// User intent pass-through into the shadow operational layer
GVL_COMMAND_SHADOW.G_Gate_Open := GVL_INTENT_USER.I_Gate_Open_Request;
GVL_COMMAND_SHADOW.G_Wicket_Open := GVL_INTENT_USER.I_Wicket_Open_Request;
GVL_COMMAND_SHADOW.G_Lock_1_Open := GVL_INTENT_USER.I_Lock_1_Open_Request;
GVL_COMMAND_SHADOW.G_Lock_1_Close := GVL_INTENT_USER.I_Lock_1_Close_Request;
GVL_COMMAND_SHADOW.G_Lock_2_Open := GVL_INTENT_USER.I_Lock_2_Open_Request;
GVL_COMMAND_SHADOW.G_Lock_2_Close := GVL_INTENT_USER.I_Lock_2_Close_Request;

// Safety and system arbitration into the shadow operational layer
IF GVL_INTENT_SAFETY.I_Fire_Alarm_Active THEN
    GVL_COMMAND_SHADOW.G_Boiler_Stop := TRUE;
    GVL_COMMAND_SHADOW.G_Vent_Stop := TRUE;
    GVL_COMMAND_SHADOW.G_Lock_1_Open := TRUE;
    GVL_COMMAND_SHADOW.G_Lock_2_Open := TRUE;
END_IF;

IF GVL_INTENT_SAFETY.I_Gas_Close_Required THEN
    GVL_COMMAND_SHADOW.G_Gas_Valve_Close := TRUE;
    GVL_COMMAND_SHADOW.G_Boiler_Stop := TRUE;
END_IF;

IF GVL_INTENT_SAFETY.I_Vent_Force_PV3_Boost THEN
    GVL_COMMAND_SHADOW.G_Vent_PV3_Boost := TRUE;
END_IF;

IF GVL_INTENT_SAFETY.I_Vent_Force_Supply_100 THEN
    GVL_COMMAND_SHADOW.G_Supply_100_Req := TRUE;
END_IF;

IF GVL_INTENT_SAFETY.I_Vent_Force_Supply_80 THEN
    GVL_COMMAND_SHADOW.G_Supply_80_Req := TRUE;
END_IF;

IF GVL_INTENT_SAFETY.I_Vent_Stop_Required THEN
    GVL_COMMAND_SHADOW.G_Vent_Stop := TRUE;
END_IF;

IF GVL_INTENT_SYSTEM.I_Mode_Degraded_Active THEN
    GVL_COMMAND_SHADOW.G_Supply_80_Req := TRUE;
END_IF;

IF GVL_INTENT_SAFETY.I_Water_Main_Close_Required THEN
    GVL_COMMAND_SHADOW.G_Close_Valve_35 := TRUE;
    GVL_COMMAND_SHADOW.G_Close_Valve_36 := TRUE;
END_IF;

FOR L_i := 1 TO 32 DO
    IF GVL_INTENT_SAFETY.I_Water_Zone_Close_Required[L_i] THEN
        ;
    END_IF;
END_FOR;
          
END_PROGRAM

PROGRAM PRG_System_Test_Harness
  VAR
    L_i : INT;
    L_j : INT;
    L_Used : REAL;
    L_HP_Used : REAL;
    L_HP_Manifold_Adjusted : ARRAY[1..GVL_CONSTANTS.C_MAX_MANIFOLDS] OF INT;
    fbDecisionTest : FB_Heating_Decision_Context;
    fbDecisionHP : FB_Heating_Decision_Context;
    fbTestResult : FB_Test_Result_Handler;
    fbTrace : FB_Trace_Logger;
  END_VAR

            IF NOT GVL_TEST.G_Test_Enable THEN
    RETURN;
END_IF;

GVL_TEST.G_Test_Total_Checks := 0;
GVL_TEST.G_Test_Failed_Checks := 0;
GVL_TEST.G_Test_Passed := TRUE;
GVL_TEST.G_Test_Last_Failure_Index := 0;
GVL_TEST.G_Test_Last_Failure_Code := 0;

// Reset transient failure flags for this scan
GVL_TEST.G_Diagnostics_Duplicate_Event_Found := FALSE;
GVL_TEST.G_Diagnostics_Count_Out_Of_Range := FALSE;
GVL_TEST.G_Heating_Allocation_Budget_Exceeded := FALSE;
GVL_TEST.G_Heating_Allocation_Enabled_Not_Allowed := FALSE;
GVL_TEST.G_Safety_Latched_Without_Intent := FALSE;
GVL_TEST.G_HP_Adjusted_Priority_Lower_Bound_Violation := FALSE;
GVL_TEST.G_HP_Adjusted_Allocation_Budget_Exceeded := FALSE;
GVL_TEST.G_HP_Adjusted_Allocation_Enabled_Not_Allowed := FALSE;
GVL_TEST.G_HP_Guest_Preheat_Config_Out_Of_Range := FALSE;

// =========================
// TEST 1: Diagnostics count bounds
// =========================
GVL_TEST.G_Test_Total_Checks := GVL_TEST.G_Test_Total_Checks + 1;
IF (GVL_STATUS.G_Diagnostics_Count < 0) OR (GVL_STATUS.G_Diagnostics_Count > 50) THEN
    GVL_TEST.G_Diagnostics_Count_Out_Of_Range := TRUE;
    GVL_TEST.G_Test_Failed_Checks := GVL_TEST.G_Test_Failed_Checks + 1;
    GVL_TEST.G_Test_Passed := FALSE;
    GVL_TEST.G_Test_Last_Failure_Index := 1;
    GVL_TEST.G_Test_Last_Failure_Code := 1001;
END_IF;

// =========================
// TEST 2: Diagnostics duplicates
// =========================
GVL_TEST.G_Test_Total_Checks := GVL_TEST.G_Test_Total_Checks + 1;
FOR L_i := 1 TO GVL_STATUS.G_Diagnostics_Count DO
    FOR L_j := L_i + 1 TO GVL_STATUS.G_Diagnostics_Count DO
        IF (GVL_STATUS.G_Diagnostics_Events[L_i].Code = GVL_STATUS.G_Diagnostics_Events[L_j].Code) AND
           (GVL_STATUS.G_Diagnostics_Events[L_i].Source = GVL_STATUS.G_Diagnostics_Events[L_j].Source) THEN
            GVL_TEST.G_Diagnostics_Duplicate_Event_Found := TRUE;
            GVL_TEST.G_Test_Failed_Checks := GVL_TEST.G_Test_Failed_Checks + 1;
            GVL_TEST.G_Test_Passed := FALSE;
            GVL_TEST.G_Test_Last_Failure_Index := 2;
            GVL_TEST.G_Test_Last_Failure_Code := 1002;
        END_IF;
    END_FOR;
END_FOR;

// =========================
// TEST 3: Base heating decision consistency
// =========================
GVL_TEST.G_Test_Total_Checks := GVL_TEST.G_Test_Total_Checks + 1;
fbDecisionTest(
    VI_Manifold_Pump_In_Service := GVL_CONFIG.G_Manifold_Pump_In_Service,
    VI_Manifold_Pressure_Fault := GVL_STATUS.G_Diagnostics.Manifold_Pressure_Fault,
    VI_Manifold_Current_Fault := GVL_STATUS.G_Diagnostics.Manifold_Current_Fault,
    VI_Manifold_Thermal_Weight := GVL_CONFIG.G_Manifold_Thermal_Weight,
    VI_Manifold_Priority := GVL_CONFIG.G_Manifold_Priority,
    VI_Max_Thermal_Budget := GVL_CONFIG.G_Max_Thermal_Budget
);

L_Used := 0.0;
FOR L_i := 1 TO GVL_CONSTANTS.C_MAX_MANIFOLDS DO
    IF fbDecisionTest.VO_Manifold_Enabled[L_i] AND (NOT fbDecisionTest.VO_Manifold_Allowed[L_i]) THEN
        GVL_TEST.G_Heating_Allocation_Enabled_Not_Allowed := TRUE;
        GVL_TEST.G_Test_Failed_Checks := GVL_TEST.G_Test_Failed_Checks + 1;
        GVL_TEST.G_Test_Passed := FALSE;
        GVL_TEST.G_Test_Last_Failure_Index := 3;
        GVL_TEST.G_Test_Last_Failure_Code := 1003;
    END_IF;

    IF fbDecisionTest.VO_Manifold_Enabled[L_i] THEN
        L_Used := L_Used + GVL_CONFIG.G_Manifold_Thermal_Weight[L_i];
    END_IF;
END_FOR;

IF L_Used > (GVL_CONFIG.G_Max_Thermal_Budget + 0.001) THEN
    GVL_TEST.G_Heating_Allocation_Budget_Exceeded := TRUE;
    GVL_TEST.G_Test_Failed_Checks := GVL_TEST.G_Test_Failed_Checks + 1;
    GVL_TEST.G_Test_Passed := FALSE;
    GVL_TEST.G_Test_Last_Failure_Index := 3;
    GVL_TEST.G_Test_Last_Failure_Code := 1004;
END_IF;

// =========================
// TEST 4: Safety latch consistency
// =========================
GVL_TEST.G_Test_Total_Checks := GVL_TEST.G_Test_Total_Checks + 1;
IF GVL_STATE.G_Safety_Gas_Latched AND (NOT GVL_INTENT_SAFETY.I_Gas_Alarm_Active) THEN
    GVL_TEST.G_Safety_Latched_Without_Intent := TRUE;
    GVL_TEST.G_Test_Failed_Checks := GVL_TEST.G_Test_Failed_Checks + 1;
    GVL_TEST.G_Test_Passed := FALSE;
    GVL_TEST.G_Test_Last_Failure_Index := 4;
    GVL_TEST.G_Test_Last_Failure_Code := 1005;
END_IF;

// =========================
// TEST 5: HP policy adjusted priority
// =========================
GVL_TEST.G_Test_Total_Checks := GVL_TEST.G_Test_Total_Checks + 1;

IF (GVL_HEATING_POLICY_CONFIG.G_Guest_Preheat_Priority_Boost < 0) OR (GVL_HEATING_POLICY_CONFIG.G_Guest_Preheat_Priority_Boost > 10) THEN
    GVL_TEST.G_HP_Guest_Preheat_Config_Out_Of_Range := TRUE;
    GVL_TEST.G_Test_Failed_Checks := GVL_TEST.G_Test_Failed_Checks + 1;
    GVL_TEST.G_Test_Passed := FALSE;
    GVL_TEST.G_Test_Last_Failure_Index := 5;
    GVL_TEST.G_Test_Last_Failure_Code := 1007;
END_IF;

FOR L_i := 1 TO GVL_CONSTANTS.C_MAX_MANIFOLDS DO
    L_HP_Manifold_Adjusted[L_i] := GVL_CONFIG.G_Manifold_Priority[L_i];
END_FOR;

FOR L_i := 1 TO GVL_CONSTANTS.C_MAX_HEATING_CIRCUITS DO
    L_j := TO_INT(GVL_CONFIG.G_HMI_FloorHeating_Configs[L_i].manifold_id);

    IF (L_j >= 1) AND (L_j <= GVL_CONSTANTS.C_MAX_MANIFOLDS) THEN
        L_HP_Manifold_Adjusted[L_j] := L_HP_Manifold_Adjusted[L_j] + TO_INT(GVL_HEATING_POLICY.G_Zone_Priority_Bias[L_i]);

        IF GVL_HEATING_POLICY_CONFIG.G_Guest_Preheat_Enabled AND GVL_HEATING_POLICY.G_Zone_Guest_Preheat_Request[L_i] THEN
            L_HP_Manifold_Adjusted[L_j] := L_HP_Manifold_Adjusted[L_j] + GVL_HEATING_POLICY_CONFIG.G_Guest_Preheat_Priority_Boost;
        END_IF;

        IF L_HP_Manifold_Adjusted[L_j] < 1 THEN
            GVL_TEST.G_HP_Adjusted_Priority_Lower_Bound_Violation := TRUE;
            GVL_TEST.G_Test_Failed_Checks := GVL_TEST.G_Test_Failed_Checks + 1;
            GVL_TEST.G_Test_Passed := FALSE;
            GVL_TEST.G_Test_Last_Failure_Index := 5;
            GVL_TEST.G_Test_Last_Failure_Code := 1006;
        END_IF;
    END_IF;
END_FOR;

FOR L_i := 1 TO GVL_CONSTANTS.C_MAX_MANIFOLDS DO
    GVL_TEST.G_HP_Manifold_Adjusted_Priority[L_i] := L_HP_Manifold_Adjusted[L_i];
END_FOR;

fbDecisionHP(
    VI_Manifold_Pump_In_Service := GVL_CONFIG.G_Manifold_Pump_In_Service,
    VI_Manifold_Pressure_Fault := GVL_STATUS.G_Diagnostics.Manifold_Pressure_Fault,
    VI_Manifold_Current_Fault := GVL_STATUS.G_Diagnostics.Manifold_Current_Fault,
    VI_Manifold_Thermal_Weight := GVL_CONFIG.G_Manifold_Thermal_Weight,
    VI_Manifold_Priority := L_HP_Manifold_Adjusted,
    VI_Max_Thermal_Budget := GVL_CONFIG.G_Max_Thermal_Budget
);

L_HP_Used := 0.0;
FOR L_i := 1 TO GVL_CONSTANTS.C_MAX_MANIFOLDS DO
    IF fbDecisionHP.VO_Manifold_Enabled[L_i] AND (NOT fbDecisionHP.VO_Manifold_Allowed[L_i]) THEN
        GVL_TEST.G_HP_Adjusted_Allocation_Enabled_Not_Allowed := TRUE;
        GVL_TEST.G_Test_Failed_Checks := GVL_TEST.G_Test_Failed_Checks + 1;
        GVL_TEST.G_Test_Passed := FALSE;
        GVL_TEST.G_Test_Last_Failure_Index := 5;
        GVL_TEST.G_Test_Last_Failure_Code := 1008;
    END_IF;

    IF fbDecisionHP.VO_Manifold_Enabled[L_i] THEN
        L_HP_Used := L_HP_Used + GVL_CONFIG.G_Manifold_Thermal_Weight[L_i];
    END_IF;
END_FOR;

IF L_HP_Used > (GVL_CONFIG.G_Max_Thermal_Budget + 0.001) THEN
    GVL_TEST.G_HP_Adjusted_Allocation_Budget_Exceeded := TRUE;
    GVL_TEST.G_Test_Failed_Checks := GVL_TEST.G_Test_Failed_Checks + 1;
    GVL_TEST.G_Test_Passed := FALSE;
    GVL_TEST.G_Test_Last_Failure_Index := 5;
    GVL_TEST.G_Test_Last_Failure_Code := 1009;
END_IF;

IF GVL_TEST.G_Test_Passed THEN
    GVL_TEST.G_Test_Status_Msg := 'ALL TESTS PASSED';
ELSE
    GVL_TEST.G_Test_Status_Msg := 'TEST FAILURES DETECTED';
END_IF;

fbTestResult(
    VI_Test_Passed := GVL_TEST.G_Test_Passed
);

IF NOT GVL_TEST.G_Test_Passed THEN
    fbTrace(
        VI_Event_Code := UDINT_TO_INT(GVL_TEST.G_Test_Last_Failure_Code),
        VI_System_Time := GVL_STATUS.G_System_Time_MS
    );
END_IF;
          
END_PROGRAM

PROGRAM PRG_IO_Write
  VAR
    L_i : INT;
  END_VAR

            // 2. ЗАПИСЬ ВЫХОДОВ (GVL_STATE -> GVL_IO)

// 2.1. Отопление (Термоэлектрические приводы)
FOR L_i := 1 TO 8 DO
    GVL_IO.DO_Zone_Valves[L_i] := GVL_STATE.G_Zone_Valves[L_i];
END_FOR;

// 2.2. Коллекторы (Насосы и смесительные клапаны)
FOR L_i := 1 TO GVL_CONSTANTS.C_MAX_MANIFOLDS DO
    GVL_IO.DO_Manifold_Pumps[L_i] := GVL_STATE.G_Manifold_Pumps[L_i];
    GVL_IO.AO_Manifold_Valves[L_i] := REAL_TO_UINT(GVL_STATE.G_Manifold_Valves[L_i] * 1000.0);
END_FOR;

// 2.4. Вентиляция
FOR L_i := 1 TO GVL_CONSTANTS.C_MAX_SUPPLY_FANS DO
    GVL_IO.AO_Supply_Fans[L_i] := REAL_TO_UINT(GVL_STATE.G_Supply_Fans[L_i] * 100.0);
END_FOR;
FOR L_i := 1 TO GVL_CONSTANTS.C_MAX_EXHAUST_FANS DO
    GVL_IO.AO_Exhaust_Fans[L_i] := REAL_TO_UINT(GVL_STATE.G_Exhaust_Fans[L_i] * 100.0);
END_FOR;

// 2.5. ГВС
GVL_IO.DO_DHW_Heating_Pump := GVL_STATE.G_DHW_Heating_Pump;
GVL_IO.DO_DHW_Circ_Pump := GVL_STATE.G_DHW_Circ_Pump;
IF GVL_STATUS.G_Is_Active_PLC THEN
    GVL_IO.DO_Backup_Circulation_Pump := GVL_STATE.G_Backup_Circulation_Pump;
    GVL_IO.DO_Electric_Heater_Enable := GVL_STATE.G_Electric_Heater_Enable;
ELSE
    GVL_IO.DO_Backup_Circulation_Pump := FALSE;
    GVL_IO.DO_Electric_Heater_Enable := FALSE;
END_IF;

// 2.6. Освещение и шторы
FOR L_i := 1 TO 8 DO
    GVL_IO.AO_Lighting_Levels[L_i] := BYTE_TO_UINT(GVL_STATE.G_Lighting_Levels[L_i]) * 10;
END_FOR;
FOR L_i := 1 TO GVL_CONSTANTS.C_MAX_BLINDS DO
    GVL_IO.AO_Blinds_Positions[L_i] := BYTE_TO_UINT(GVL_STATE.G_Blinds_Positions[L_i]) * 10;
END_FOR;

// 2.7. Аварийные выходы (Сирены и клапаны)
GVL_IO.DO_Gas_Siren := (GVL_ALARM.G_Gas_Fire_Siren AND GVL_ALARM.G_Gas_Alarm_Active);
GVL_IO.DO_Fire_Siren := (GVL_ALARM.G_Gas_Fire_Siren AND GVL_ALARM.G_Fire_Alarm_Active);
GVL_IO.DO_Security_Siren := GVL_ALARM.G_Security_Siren;

// === STAGE H2: USE SHADOW COMMANDS ===
GVL_IO.DO_Water_Valve_35_Close := GVL_COMMAND_SHADOW.G_Close_Valve_35;
GVL_IO.DO_Water_Valve_36_Close := GVL_COMMAND_SHADOW.G_Close_Valve_36;
GVL_IO.DO_Gas_Valve_Close := GVL_COMMAND_SHADOW.G_Gas_Valve_Close;

// Access control (shadow)
GVL_IO.DO_Lock_1_Open := GVL_COMMAND_SHADOW.G_Lock_1_Open;
GVL_IO.DO_Lock_1_Close := GVL_COMMAND_SHADOW.G_Lock_1_Close;
GVL_IO.DO_Lock_2_Open := GVL_COMMAND_SHADOW.G_Lock_2_Open;
GVL_IO.DO_Lock_2_Close := GVL_COMMAND_SHADOW.G_Lock_2_Close;

// Gate/Wicket — now via shadow
GVL_IO.DO_Gate_Open := GVL_COMMAND_SHADOW.G_Gate_Open;
GVL_IO.DO_Wicket_Open := GVL_COMMAND_SHADOW.G_Wicket_Open;

// 2.9. Розетки
GVL_IO.DO_Sockets := GVL_STATE.G_Socket_States;

// Selective zonal water recovery outputs
FOR L_i := 1 TO 32 DO
    GVL_IO.DO_Water_Zone_Enable[L_i] := GVL_STATE.G_Water_Zone_Enable[L_i];
END_FOR;

// >>> BULK_SYNC_ANCHOR: PRG_IO_Write <<<
          
END_PROGRAM

PROGRAM PRG_System
  VAR
    L_i : INT;
    L_Motion_Sensors_16 : ARRAY[1..16] OF BOOL;
    L_Zone_Valves_8 : ARRAY[1..8] OF BOOL;
    L_Lighting_32 : ARRAY[1..32] OF BYTE;
    L_Lighting_Bool_32 : ARRAY[1..32] OF BOOL;
    L_FloorTemps_8 : ARRAY[1..8] OF REAL;
    fbCoreKernelObserver : FB_CoreKernel_Live_Observer;    fbSimulationManager : FB_Simulation_Manager;
    fbRuleEngine : FB_Rule_Engine;
    fbBlackBox : FB_BlackBox_Recorder;
    fbAstroTimer : FB_Astro_Timer;    fbHistoryManager : FB_History_Manager;    fbLogEvent : FB_LogEvent;
    fbSystemScenarioArb : FB_System_Scenario_Arbitration;
    fbSystemGatewayIntent : FB_System_Gateway_Intent;
    fbSystemPersist : FB_System_Persist_Manager;
    fbSystemInit : FB_System_Init;
    fbSystemRecovery : FB_System_Recovery;
    fbTimebase : FB_System_Timebase;
    fbSystemRedundancy : FB_System_Redundancy_Orchestrator;
    fbSystemHealthOrchestrator : FB_System_Health_Orchestrator;
    fbSystemIntentPublisher : FB_System_Intent_Publisher;
    fbSystemEvacuation : FB_System_Evacuation;
    fbSystemAlarmOrchestrator : FB_System_Alarm_Orchestrator;
    L_Time_Diff : UDINT;
    L_Local_State : ST_System_State_Snapshot;
    L_Remote_State : ST_System_State_Snapshot;
    L_NVRAM_Cmd : BYTE;
    L_NVRAM_Offset : UDINT;
    L_NVRAM_Done : BOOL;
    L_NVRAM_Err : BOOL;
    L_NVRAM_ErrID : UDINT;
    L_BB_Record : ST_BlackBox_Record;
    L_BB_Freeze : BOOL;
    L_Scenario_Idx : INT;
    L_Last_Operator_Blocked : BOOL;
    L_Last_DHW_Heating_In_Service : BOOL;
    L_Last_DHW_Circ_In_Service : BOOL;
    L_Dangerous_Action_Armed : BOOL;
    L_Dangerous_Action_Deadline_MS : UDINT;
    L_Maintenance_Apply_Intent : BOOL;
    L_Last_System_Mode : E_System_Operating_Mode;
    L_Last_First_Fault_Type : INT;
    L_Last_First_Fault_Source : INT;
    L_First_Fault_Active : BOOL;
    L_First_Fault_Type : INT;
    L_First_Fault_Source : INT;
    L_System_Severity : E_System_Severity;
    L_Root_Cause : E_System_Root_Cause;
    L_Watchdog_Fault : BOOL;
    L_Last_Root_Cause : E_System_Root_Cause;
    L_History_Event : ST_History_Record;
    L_History_Write_Event : BOOL;
    L_Last_Operator_Journal_Seq : UDINT;
    L_Last_Event_Code : UDINT;
    L_Last_Event_Value : REAL;
    L_Last_Event_Time_MS : UDINT;
    L_Gateway_Writes_Allowed : BOOL;
    L_Scenario_Req_Operator : E_SCENARIO_TYPE;
    L_Scenario_Req_Gateway : E_SCENARIO_TYPE;
    L_Scenario_Req_Rule : E_SCENARIO_TYPE;
    L_Scenario_Req_Final : E_SCENARIO_TYPE;
    L_Scenario_Intent : E_SCENARIO_TYPE;
    L_Scenario_Source : E_SCENARIO_SOURCE;
    L_Scenario_Changed : BOOL;
    L_Last_Scenario_Change_Time : UDINT;
    L_IO_Fault : BOOL;
    L_IO_Fault_Prev : BOOL;
    L_Comm_Fault_Prev : BOOL;
    L_Sensor_Fault_Prev : BOOL;
    L_Subsystem_Fault_Prev : BOOL;
    L_Mode_Prev : E_System_Operating_Mode;
    L_User_Access_Denied_Prev : BOOL;
    L_Persist_Buffer : ARRAY[0..4] OF BYTE;
    L_Last_Written_Persist_Buffer : ARRAY[0..4] OF BYTE;
    L_Persist_Buffer_Changed : BOOL;
    L_Last_Persist_Write_MS : UDINT;
    L_Recovery_Done : BOOL;
    L_Persist_Struct : ST_Persist;
  END_VAR

            // 0. Инициализация RETAIN переменных при первом запуске
fbSystemInit(
    VIO_Local_State := L_Local_State,
    VIO_Remote_State := L_Remote_State
);

// === NVRAM RECOVERY (ONCE AFTER BOOT) ===
fbSystemRecovery(
    VIO_Recovery_Done := L_Recovery_Done
);

// === Persist manager ===
fbSystemPersist(
    VI_System_Time_MS := GVL_STATUS.G_System_Time_MS,
    VI_IsActivePLC := GVL_STATUS.G_Is_Active_PLC,
    VIO_Persist_Buffer := L_Persist_Buffer,
    VIO_Last_Written_Persist_Buffer := L_Last_Written_Persist_Buffer,
    VIO_Persist_Buffer_Changed := L_Persist_Buffer_Changed,
    VIO_Last_Persist_Write_MS := L_Last_Persist_Write_MS,
    VIO_NVRAM_Cmd := L_NVRAM_Cmd,
    VIO_NVRAM_Offset := L_NVRAM_Offset,
    VIO_NVRAM_Done := L_NVRAM_Done,
    VIO_NVRAM_Err := L_NVRAM_Err,
    VIO_NVRAM_ErrID := L_NVRAM_ErrID
);

// NVRAM CONTROLLED WRITE ENABLED (step 8B)

// 1. Обновление системного времени
fbTimebase();

// 2-3. Redundancy / state sync
fbSystemRedundancy(
    VIO_Local_State := L_Local_State,
    VIO_Remote_State := L_Remote_State
);

// 3.4-3.7. Safety / health / state mode
fbSystemHealthOrchestrator(
    VO_First_Fault_Active => L_First_Fault_Active,
    VO_First_Fault_Type => L_First_Fault_Type,
    VO_First_Fault_Source => L_First_Fault_Source,
    VO_System_Severity => L_System_Severity,
    VO_Root_Cause => L_Root_Cause,
    VO_Watchdog_Fault => L_Watchdog_Fault
);

// === STAGE G2b: SYSTEM GATE PUBLICATION ===
fbSystemIntentPublisher(
    VI_System_Time_MS := GVL_STATUS.G_System_Time_MS,
    VI_Gateway_Writes_Allowed := L_Gateway_Writes_Allowed
);

// 3.6a. Эвакуация
fbSystemEvacuation();

// 4. Астрономический таймер
fbAstroTimer(
    VI_System_Time_MS := GVL_STATUS.G_System_Time_MS,
    VI_Latitude := 55.75,
    VI_Longitude := 37.61,
    VI_Day_Of_Year := GVL_STATUS.G_Day_Of_Year,
    VO_Is_Night => GVL_STATUS.G_Is_Night
);


// 5. Управление сценариями
// Scenario request (direct + early operator gate)
IF GVL_STATE.G_System_Mode = E_System_Operating_Mode.MODE_NORMAL THEN
    L_Scenario_Req_Operator := GVL_COMMAND.G_Scenario_Request_Operator;
ELSE
    L_Scenario_Req_Operator := E_SCENARIO_TYPE.SCENARIO_NONE;
END_IF;
L_Scenario_Req_Gateway := 0;
L_Scenario_Req_Rule := 0;







// Синхронизируем request с фактически активным сценарием


L_Scenario_Idx := TO_INT(GVL_STATUS.G_Current_Scenario);
IF L_Scenario_Idx < 0 OR L_Scenario_Idx > 7 THEN
    L_Scenario_Idx := 0;
END_IF;

// === Scenario arbitration ===
fbSystemScenarioArb(
    VI_System_Time_MS := GVL_STATUS.G_System_Time_MS,
    VI_IsActivePLC := GVL_STATUS.G_Is_Active_PLC,
    VI_System_Mode := GVL_STATE.G_System_Mode,
    VI_Security_Armed := GVL_ALARM.G_Security_Armed,
    VIO_Scenario_Req_Operator := L_Scenario_Req_Operator,
    VIO_Scenario_Req_Gateway := L_Scenario_Req_Gateway,
    VIO_Scenario_Req_Rule := L_Scenario_Req_Rule,
    VIO_Scenario_Req_Final := L_Scenario_Req_Final,
    VIO_Scenario_Intent := L_Scenario_Intent,
    VIO_Scenario_Source := L_Scenario_Source
);

// 6. Симуляция присутствия
fbSimulationManager(
    VI_System_Time_MS := GVL_STATUS.G_System_Time_MS,
    VI_IsActivePLC := GVL_STATUS.G_Is_Active_PLC AND (GVL_STATE.G_System_Mode = E_System_Operating_Mode.MODE_NORMAL),
    VI_Scenario := GVL_STATUS.G_Current_Scenario,
    VI_Config := GVL_CONFIG.G_HMI_Scenario_Configs[L_Scenario_Idx],
    VO_Sim_Lights => GVL_STATE.G_Sim_Lights,
    VO_Sim_Active => GVL_STATUS.G_Sim_Active
);

// 6.5. Пользовательские правила (Rule Engine)
fbRuleEngine(
    VI_System_Time_MS := GVL_STATUS.G_System_Time_MS,
    VI_IsActivePLC := GVL_STATUS.G_Is_Active_PLC,
    VI_Rules := GVL_CONFIG.G_HMI_User_Rules,
    VI_Indoor_Temps := GVL_STATE.G_Room_Temps,
    VI_Floor_Temps := L_FloorTemps_8,
    VI_Humidities := GVL_STATE.G_Room_Hum,
    VI_CO2_Levels := GVL_STATE.G_Room_CO2,
    VI_Motion_Sensors := L_Motion_Sensors_16,
    VI_Door_Sensors := GVL_STATE.G_Door_Sensors,
    VI_Window_Sensors := GVL_STATE.G_Window_Sensors,
    VI_Water_Sensors := GVL_STATE.G_Water_Sensors,
    VI_Smoke_Sensors := GVL_STATE.G_Smoke_Sensors,
    VI_Methane_Sensors := GVL_STATE.G_Methane_Sensors,
    VI_CO_Sensors := GVL_STATE.G_CO_Sensors,
    VI_Security_Armed := GVL_ALARM.G_Security_Armed,
    VI_Current_Time := GVL_STATUS.G_Current_TOD,
    VI_Day_Of_Week := TO_INT(GVL_STATUS.G_Current_Day),
    VO_Actions => GVL_STATE.G_Rule_Actions
);

FOR L_i := 1 TO GVL_CONSTANTS.C_MAX_RULES DO
    IF GVL_STATE.G_Rule_Actions[L_i].Active AND GVL_STATE.G_Rule_Actions[L_i].Action_Type = E_Rule_Action_Type.ACTION_ACTIVATE_SCENARIO THEN
        L_Scenario_Req_Rule := TO_BYTE(GVL_STATE.G_Rule_Actions[L_i].Value);
    END_IF;
END_FOR;



// 8.5 Менеджер тревог
fbSystemAlarmOrchestrator(
    VI_First_Fault_Active := L_First_Fault_Active,
    VI_First_Fault_Type := L_First_Fault_Type,
    VI_First_Fault_Source := L_First_Fault_Source
);

// Command arbitration: OPERATOR > GATEWAY
L_Gateway_Writes_Allowed :=
    NOT GVL_STATUS.G_Diagnostics.Dangerous_Action_Pending_Confirm AND
    NOT GVL_STATUS.G_Diagnostics.Operator_Action_Blocked AND
    NOT GVL_STATUS.G_Diagnostics.User_Access_Denied;

// === Gateway intent ===
fbSystemGatewayIntent(
    VI_System_Time_MS := GVL_STATUS.G_System_Time_MS,
    VI_IsActivePLC := GVL_STATUS.G_Is_Active_PLC,
    VI_Gateway_Writes_Allowed := L_Gateway_Writes_Allowed,
    VIO_FloorHeating_Temps := L_FloorTemps_8,
    VIO_Zone_Valve_States := L_Zone_Valves_8,
    VIO_Lighting_Base_Levels := L_Lighting_32,
    VIO_Scenario_Req_Gateway := L_Scenario_Req_Gateway
);

// Gateway moved to helper

// Persist/NVRAM moved to helper

// 15. Черный ящик
L_BB_Record.Timestamp := GVL_STATUS.G_System_Time_MS;
L_BB_Record.PLC_Active_ID := GVL_STATUS.G_PLC_ID;
L_BB_Record.Gas_Methane_LEL := GVL_STATE.G_Methane_Sensors[1];
L_BB_Record.Gas_CO_PPM := GVL_STATE.G_CO_Sensors[1];
L_BB_Record.Flood_Active := GVL_ALARM.G_Flood_Alarm_Active;
L_BB_Record.Fire_Active := GVL_ALARM.G_Fire_Alarm_Active;
L_BB_Record.Valve_Gas_Status := SEL(GVL_COMMAND.G_Gas_Valve_Close, BYTE#0, BYTE#1);
L_BB_Record.Valve_Water_Status := SEL((GVL_COMMAND.G_Close_Valve_35 OR GVL_COMMAND.G_Close_Valve_36), BYTE#0, BYTE#1);

L_BB_Record.System_Mode := TO_BYTE(TO_INT(GVL_STATE.G_System_Mode));
L_BB_Record.First_Fault_Type := TO_BYTE(TO_INT(L_First_Fault_Type));
L_BB_Record.First_Fault_Source := TO_BYTE(TO_INT(L_First_Fault_Source));
L_BB_Record.First_Fault_Active := L_First_Fault_Active;
L_BB_Record.System_Severity := TO_BYTE(TO_INT(L_System_Severity));
L_BB_Record.Root_Cause := TO_BYTE(TO_INT(L_Root_Cause));
L_BB_Record.Watchdog_Fault := L_Watchdog_Fault;


L_BB_Freeze := GVL_ALARM.G_Gas_Alarm_Active OR GVL_ALARM.G_Fire_Alarm_Active OR GVL_ALARM.G_Flood_Alarm_Active OR L_First_Fault_Active;

fbBlackBox(
    VI_Current_Data := L_BB_Record,
    VI_Freeze := L_BB_Freeze
);

// 15.1. Менеджер истории / diagnostics bridge
L_History_Write_Event := FALSE;
L_History_Event.timestamp_ms := GVL_STATUS.G_System_Time_MS;
L_History_Event.event_code := 0;
L_History_Event.event_value := 0.0;
L_History_Event.unit := 0;
L_History_Event.zone_id := 0;
L_History_Event.operator_id := 'SYSTEM';
L_History_Event.priority := E_ALERT_PRIORITY.ALERT_PRIORITY_HIGH;

IF GVL_STATE.G_System_Mode <> L_Last_System_Mode THEN
    L_History_Write_Event := TRUE;
    L_History_Event.event_code := 1101; // System mode transition
    L_History_Event.event_value := TO_REAL(TO_INT(GVL_STATE.G_System_Mode));
    L_History_Event.unit := 1; // system mode domain
    L_History_Event.zone_id := 0;
    IF GVL_STATE.G_System_Mode = E_System_Operating_Mode.MODE_NORMAL THEN
        L_History_Event.priority := E_ALERT_PRIORITY.ALERT_PRIORITY_HIGH;
    ELSE
        L_History_Event.priority := E_ALERT_PRIORITY.ALERT_PRIORITY_HIGH;
    END_IF;
    L_Last_System_Mode := GVL_STATE.G_System_Mode;

ELSIF L_Root_Cause <> L_Last_Root_Cause THEN
    L_History_Write_Event := TRUE;
    L_History_Event.event_code := 1102; // Root cause changed
    L_History_Event.event_value := TO_REAL(TO_INT(L_Root_Cause));
    L_History_Event.unit := 2; // root cause enum domain
    L_History_Event.zone_id := TO_BYTE(L_First_Fault_Source);
    L_History_Event.priority := E_ALERT_PRIORITY.ALERT_PRIORITY_HIGH;
    L_Last_Root_Cause := L_Root_Cause;

ELSIF L_First_Fault_Source <> L_Last_First_Fault_Source THEN
    L_History_Write_Event := TRUE;
    L_History_Event.event_code := 1103; // First fault source changed
    L_History_Event.event_value := TO_REAL(L_First_Fault_Source);
    L_History_Event.unit := 3; // root cause source domain
    L_History_Event.zone_id := TO_BYTE(L_First_Fault_Source);
    L_History_Event.priority := E_ALERT_PRIORITY.ALERT_PRIORITY_HIGH;
    L_Last_First_Fault_Source := L_First_Fault_Source;

ELSIF GVL_STATUS.G_Current_Scenario <> GVL_STATUS.G_Previous_Scenario THEN
    L_History_Write_Event := TRUE;
    L_History_Event.event_code := 1001; // Scenario transition
    L_History_Event.event_value := TO_REAL(GVL_STATUS.G_Current_Scenario);
    L_History_Event.unit := 4; // scenario domain
    L_History_Event.zone_id := 0;
    L_History_Event.priority := E_ALERT_PRIORITY.ALERT_PRIORITY_HIGH;
    GVL_STATUS.G_Previous_Scenario := GVL_STATUS.G_Current_Scenario;

ELSIF GVL_STATUS.G_Diagnostics.Alarm_Event_Pulse THEN
    L_History_Write_Event := TRUE;
    L_History_Event.event_code := TO_WORD(GVL_STATUS.G_Diagnostics.Alarm_Event_Code);
    L_History_Event.event_value := GVL_STATUS.G_Diagnostics.Alarm_Event_Value;
    L_History_Event.unit := 10; // alarm lifecycle domain
    L_History_Event.zone_id := 0;
    L_History_Event.priority := E_ALERT_PRIORITY.ALERT_PRIORITY_HIGH;

ELSIF GVL_STATUS.G_Diagnostics.Operator_Journal_Event_Seq <> L_Last_Operator_Journal_Seq THEN
    L_History_Write_Event := TRUE;
    L_History_Event.event_code := 1301; // Operator journal event
    L_History_Event.event_value := TO_REAL(GVL_STATUS.G_Diagnostics.Operator_Journal_Event_Seq);
    L_History_Event.unit := 20; // operator journal domain
    L_History_Event.zone_id := 0;
    L_History_Event.priority := E_ALERT_PRIORITY.ALERT_PRIORITY_HIGH;
    L_Last_Operator_Journal_Seq := GVL_STATUS.G_Diagnostics.Operator_Journal_Event_Seq;
END_IF;

// --- History anti-flood / dedup ---
IF L_History_Write_Event THEN
    IF (L_History_Event.event_code = L_Last_Event_Code)
       AND (ABS(L_History_Event.event_value - L_Last_Event_Value) < 0.001)
       AND (GVL_STATUS.G_System_Time_MS - L_Last_Event_Time_MS < 5000) THEN
        L_History_Write_Event := FALSE;
    ELSE
        L_Last_Event_Code := L_History_Event.event_code;
        L_Last_Event_Value := L_History_Event.event_value;
        L_Last_Event_Time_MS := GVL_STATUS.G_System_Time_MS;
    END_IF;
END_IF;

fbHistoryManager(
    VI_System_Time_MS := GVL_STATUS.G_System_Time_MS,
    VI_Write_Event := L_History_Write_Event,
    VI_Event := L_History_Event
);


L_Maintenance_Apply_Intent := FALSE;

// Dangerous action confirmation flow
IF GVL_COMMAND.CMD_Dangerous_Action_Request AND (GVL_COMMAND.CMD_User_Access_Level >= 2) THEN

    IF NOT L_Dangerous_Action_Armed THEN
        fbLogEvent(
            VI_Event_Type := 8,
            VI_Timestamp := GVL_STATUS.G_System_Time_MS,
            VI_Param1 := TO_UDINT(GVL_COMMAND.CMD_User_Access_Level),
            VI_Param2 := 1
        );
    END_IF;

    L_Dangerous_Action_Armed := TRUE;
    L_Dangerous_Action_Deadline_MS := GVL_STATUS.G_System_Time_MS + 15000;
    GVL_STATUS.G_Diagnostics.Dangerous_Action_Pending_Confirm := TRUE;
    GVL_STATUS.G_Diagnostics.Dangerous_Action_Confirm_Deadline_MS := L_Dangerous_Action_Deadline_MS;
    GVL_STATUS.G_Diagnostics.Dangerous_Action_Confirm_Text := 'Подтвердите опасное действие в течение 15 секунд';
END_IF;
IF L_Dangerous_Action_Armed AND (GVL_STATUS.G_System_Time_MS > L_Dangerous_Action_Deadline_MS) THEN
    L_Dangerous_Action_Armed := FALSE;
    GVL_STATUS.G_Diagnostics.Dangerous_Action_Pending_Confirm := FALSE;
    GVL_STATUS.G_Diagnostics.Dangerous_Action_Confirm_Text := 'Окно подтверждения истекло';
END_IF;
IF GVL_COMMAND.CMD_Dangerous_Action_Confirm AND
   L_Dangerous_Action_Armed AND
   (GVL_COMMAND.CMD_User_Access_Level >= 2) THEN
    L_Maintenance_Apply_Intent := TRUE;

    fbLogEvent(
        VI_Event_Type := 9,
        VI_Timestamp := GVL_STATUS.G_System_Time_MS,
        VI_Param1 := TO_UDINT(GVL_COMMAND.CMD_User_Access_Level),
        VI_Param2 := 1
    );

    L_Dangerous_Action_Armed := FALSE;
    GVL_STATUS.G_Diagnostics.Dangerous_Action_Pending_Confirm := FALSE;
    GVL_STATUS.G_Diagnostics.Dangerous_Action_Confirm_Text := 'Опасное действие подтверждено оператором';
END_IF;

// HMI maintenance mode control (confirmation-aware)
IF L_Maintenance_Apply_Intent THEN
    FOR L_i := 1 TO GVL_CONSTANTS.C_MAX_MANIFOLDS DO
        GVL_CONFIG.G_Manifold_Pump_In_Service[L_i] := GVL_COMMAND.CMD_Set_Manifold_Pump_In_Service[L_i];
    END_FOR;
    GVL_CONFIG.G_DHW_Heating_Pump_In_Service := GVL_COMMAND.CMD_Set_DHW_Heating_Pump_In_Service;
    GVL_CONFIG.G_DHW_Circ_Pump_In_Service := GVL_COMMAND.CMD_Set_DHW_Circ_Pump_In_Service;
END_IF;

// Access level enforcement for dangerous actions
GVL_STATUS.G_Diagnostics.User_Access_Level_Active := GVL_COMMAND.CMD_User_Access_Level;
GVL_STATUS.G_Diagnostics.User_Access_Denied := FALSE;
GVL_STATUS.G_Diagnostics.User_Access_Deny_Reason := '';
IF GVL_COMMAND.CMD_Dangerous_Action_Request OR GVL_COMMAND.CMD_Dangerous_Action_Confirm THEN
    IF GVL_COMMAND.CMD_User_Access_Level < 2 THEN
        IF NOT L_User_Access_Denied_Prev THEN
            fbLogEvent(
                VI_Event_Type := 10,
                VI_Timestamp := GVL_STATUS.G_System_Time_MS,
                VI_Param1 := TO_UDINT(GVL_COMMAND.CMD_User_Access_Level),
                VI_Param2 := 2
            );
        END_IF;

        GVL_STATUS.G_Diagnostics.User_Access_Denied := TRUE;
        GVL_STATUS.G_Diagnostics.User_Access_Deny_Reason := 'Недостаточный уровень доступа для опасного действия';
        GVL_STATUS.G_Diagnostics.Operator_Action_Blocked := TRUE;
        GVL_STATUS.G_Diagnostics.Operator_Block_Reason := 'Требуется уровень ENGINEER для опасного действия';
        GVL_STATUS.G_Diagnostics.Dangerous_Action_Pending_Confirm := FALSE;
        GVL_STATUS.G_Diagnostics.Dangerous_Action_Confirm_Text := 'Доступ запрещён: требуется уровень ENGINEER';
    END_IF;
END_IF;

L_User_Access_Denied_Prev := GVL_STATUS.G_Diagnostics.User_Access_Denied;

// Hard revert for forbidden operator actions
IF GVL_STATUS.G_Diagnostics.Operator_Action_Blocked THEN
    FOR L_i := 1 TO GVL_CONSTANTS.C_MAX_MANIFOLDS DO
        IF NOT GVL_CONFIG.G_Manifold_Pump_In_Service[L_i] THEN
            GVL_CONFIG.G_Manifold_Pump_In_Service[L_i] := TRUE;
        END_IF;
    END_FOR;
    IF NOT GVL_CONFIG.G_DHW_Heating_Pump_In_Service THEN
        GVL_CONFIG.G_DHW_Heating_Pump_In_Service := TRUE;
    END_IF;
    IF NOT GVL_CONFIG.G_DHW_Circ_Pump_In_Service THEN
        GVL_CONFIG.G_DHW_Circ_Pump_In_Service := TRUE;
    END_IF;
    GVL_STATUS.G_Diagnostics.Operator_Last_Forbidden_Action := GVL_STATUS.G_Diagnostics.Operator_Block_Reason;
END_IF;

// Operator action journal
IF GVL_STATUS.G_Diagnostics.Operator_Action_Blocked AND NOT L_Last_Operator_Blocked THEN
    GVL_STATUS.G_Diagnostics.Operator_Journal_Event_Seq := GVL_STATUS.G_Diagnostics.Operator_Journal_Event_Seq + 1;
END_IF;
L_Last_Operator_Blocked := GVL_STATUS.G_Diagnostics.Operator_Action_Blocked;
IF GVL_CONFIG.G_DHW_Heating_Pump_In_Service <> L_Last_DHW_Heating_In_Service THEN
    GVL_STATUS.G_Diagnostics.Operator_Journal_Event_Seq := GVL_STATUS.G_Diagnostics.Operator_Journal_Event_Seq + 1;
    IF GVL_CONFIG.G_DHW_Heating_Pump_In_Service THEN
        GVL_STATUS.G_Diagnostics.Maintenance_Last_Action := 'Насос загрузки ГВС возвращён из ТО';
    ELSE
        GVL_STATUS.G_Diagnostics.Maintenance_Last_Action := 'Насос загрузки ГВС выведен в ТО';
    END_IF;
END_IF;
L_Last_DHW_Heating_In_Service := GVL_CONFIG.G_DHW_Heating_Pump_In_Service;
IF GVL_CONFIG.G_DHW_Circ_Pump_In_Service <> L_Last_DHW_Circ_In_Service THEN
    GVL_STATUS.G_Diagnostics.Operator_Journal_Event_Seq := GVL_STATUS.G_Diagnostics.Operator_Journal_Event_Seq + 1;
    IF GVL_CONFIG.G_DHW_Circ_Pump_In_Service THEN
        GVL_STATUS.G_Diagnostics.Maintenance_Last_Action := 'Насос рециркуляции ГВС возвращён из ТО';
    ELSE
        GVL_STATUS.G_Diagnostics.Maintenance_Last_Action := 'Насос рециркуляции ГВС выведен в ТО';
    END_IF;
END_IF;
L_Last_DHW_Circ_In_Service := GVL_CONFIG.G_DHW_Circ_Pump_In_Service;
IF GVL_STATUS.G_Diagnostics.Operator_Journal_Event_Seq <> GVL_STATUS.G_Diagnostics.Operator_Journal_Last_Seq THEN
    GVL_STATUS.G_Diagnostics.Operator_Journal_3 := GVL_STATUS.G_Diagnostics.Operator_Journal_2;
    GVL_STATUS.G_Diagnostics.Operator_Journal_2 := GVL_STATUS.G_Diagnostics.Operator_Journal_1;
    IF GVL_STATUS.G_Diagnostics.Operator_Last_Forbidden_Action <> '' THEN
        GVL_STATUS.G_Diagnostics.Operator_Journal_1 := GVL_STATUS.G_Diagnostics.Operator_Last_Forbidden_Action;
    ELSE
        GVL_STATUS.G_Diagnostics.Operator_Journal_1 := GVL_STATUS.G_Diagnostics.Maintenance_Last_Action;
    END_IF;
    GVL_STATUS.G_Diagnostics.Operator_Journal_Last_Seq := GVL_STATUS.G_Diagnostics.Operator_Journal_Event_Seq;
END_IF;

// ========================================
// CoreKernel live observer (diagnostic only)
// ========================================
// fbCoreKernelObserver disabled temporarily


// === NVRAM SNAPSHOT VIA STRUCT ADAPTER ===
L_Persist_Struct.System_Mode := GVL_STATE.G_System_Mode;

L_Persist_Struct.Safety_Gas_Latched := GVL_STATE.G_Safety_Gas_Latched;
L_Persist_Struct.Safety_Smoke_Latched := GVL_STATE.G_Safety_Smoke_Latched;
L_Persist_Struct.Safety_Leak_Latched := GVL_STATE.G_Safety_Leak_Latched;

L_Persist_Struct.DHW_Heating_Pump := GVL_STATE.G_DHW_Heating_Pump;
L_Persist_Struct.Valid := TRUE;

// mirror to legacy persistent variables
GVL_PERSISTENT.P_System_Mode := L_Persist_Struct.System_Mode;

GVL_PERSISTENT.P_Safety_Gas_Latched := L_Persist_Struct.Safety_Gas_Latched;
GVL_PERSISTENT.P_Safety_Smoke_Latched := L_Persist_Struct.Safety_Smoke_Latched;
GVL_PERSISTENT.P_Safety_Leak_Latched := L_Persist_Struct.Safety_Leak_Latched;

GVL_PERSISTENT.P_DHW_Heating_Active := L_Persist_Struct.DHW_Heating_Pump;
GVL_PERSISTENT.P_Valid := L_Persist_Struct.Valid;

// >>> BULK_SYNC_ANCHOR: PRG_System <<<

// === EVENT LOGGING: SCENARIO CHANGE ===
IF L_Scenario_Changed THEN
    fbLogEvent(
        VI_Event_Type := 1,
        VI_Timestamp := GVL_STATUS.G_System_Time_MS,
        VI_Param1 := TO_UDINT(L_Scenario_Source),
        VI_Param2 := TO_UDINT(L_Scenario_Intent)
    );
END_IF;

// === EVENT LOGGING: FAULTS ===

// IO
IF GVL_STATUS.G_Diagnostics.IO_Offline AND NOT L_IO_Fault_Prev THEN
    fbLogEvent(
        VI_Event_Type := 2,
        VI_Timestamp := GVL_STATUS.G_System_Time_MS,
        VI_Param1 := 1,
        VI_Param2 := 1
    );
END_IF;

IF NOT GVL_STATUS.G_Diagnostics.IO_Offline AND L_IO_Fault_Prev THEN
    fbLogEvent(
        VI_Event_Type := 3,
        VI_Timestamp := GVL_STATUS.G_System_Time_MS,
        VI_Param1 := 1,
        VI_Param2 := 0
    );
END_IF;

L_IO_Fault_Prev := GVL_STATUS.G_Diagnostics.IO_Offline;

// === EVENT LOGGING: MODE CHANGE ===
IF GVL_STATE.G_System_Mode <> L_Mode_Prev THEN
    fbLogEvent(
        VI_Event_Type := 4,
        VI_Timestamp := GVL_STATUS.G_System_Time_MS,
        VI_Param1 := TO_UDINT(L_Mode_Prev),
        VI_Param2 := TO_UDINT(GVL_STATE.G_System_Mode)
    );
END_IF;

L_Mode_Prev := GVL_STATE.G_System_Mode;
          
END_PROGRAM

PROGRAM PRG_Test_Scenario_Runner

            IF NOT GVL_TEST.G_Test_Enable THEN
    RETURN;
END_IF;

IF NOT GVL_TEST_INJECTION.G_Scenario_Enable THEN
    RETURN;
END_IF;

// Reset request
IF GVL_TEST_INJECTION.G_Scenario_Reset_Request THEN
    GVL_TEST_INJECTION.G_Inject_Enable := FALSE;
    GVL_TEST_INJECTION.G_Inject_Gas_Level := 0.0;
    GVL_TEST_INJECTION.G_Inject_Force_Gas_Alarm_Reset := FALSE;
    GVL_TEST_INJECTION.G_Inject_Force_IO_Offline := FALSE;
    GVL_TEST_INJECTION.G_Scenario_Step := 0;
    GVL_TEST_INJECTION.G_Scenario_Done := FALSE;
    GVL_TEST_INJECTION.G_Scenario_Failed := FALSE;
    GVL_TEST_INJECTION.G_Scenario_Reset_Request := FALSE;
END_IF;

CASE GVL_TEST_INJECTION.G_Scenario_Current OF

// =========================
// SCENARIO 1: GAS + WATCHDOG
// =========================
1:
    CASE GVL_TEST_INJECTION.G_Scenario_Step OF
    0:
        GVL_TEST_INJECTION.G_Inject_Enable := TRUE;
        GVL_TEST_INJECTION.G_Inject_Gas_Level := 50.0;
        GVL_TEST_INJECTION.G_Scenario_Status_Msg := 'Gas injected';
        GVL_TEST_INJECTION.G_Scenario_Step := 1;

    1:
        GVL_TEST_INJECTION.G_Inject_Force_Gas_Alarm_Reset := TRUE;
        GVL_TEST_INJECTION.G_Scenario_Status_Msg := 'Forced alarm reset';
        GVL_TEST_INJECTION.G_Scenario_Step := 2;

    2:
        IF GVL_TEST.G_Ownership_Violation THEN
            GVL_TEST_INJECTION.G_Scenario_Done := TRUE;
            GVL_TEST_INJECTION.G_Scenario_Status_Msg := 'Watchdog OK';
        ELSE
            GVL_TEST_INJECTION.G_Scenario_Failed := TRUE;
        END_IF;
    END_CASE;

// =========================
// SCENARIO 2: IO OFFLINE
// =========================
2:
    CASE GVL_TEST_INJECTION.G_Scenario_Step OF
    0:
        GVL_TEST_INJECTION.G_Inject_Enable := TRUE;
        GVL_TEST_INJECTION.G_Inject_Force_IO_Offline := TRUE;
        GVL_TEST_INJECTION.G_Scenario_Status_Msg := 'IO offline injected';
        GVL_TEST_INJECTION.G_Scenario_Step := 1;

    1:
        IF NOT GVL_STATUS.G_IO_Modules_Online[1] THEN
            GVL_TEST_INJECTION.G_Scenario_Done := TRUE;
            GVL_TEST_INJECTION.G_Scenario_Status_Msg := 'IO fail-safe OK';
        ELSE
            GVL_TEST_INJECTION.G_Scenario_Failed := TRUE;
        END_IF;
    END_CASE;

END_CASE;

// Auto advance
IF GVL_TEST_INJECTION.G_Scenario_Done AND GVL_TEST_INJECTION.G_Scenario_Auto_Run THEN
    GVL_TEST_INJECTION.G_Scenario_Current := GVL_TEST_INJECTION.G_Scenario_Current + 1;
    GVL_TEST_INJECTION.G_Scenario_Reset_Request := TRUE;
END_IF;
          
END_PROGRAM

PROGRAM PRG_Ventilation
  VAR
    fbVentilationManager : FB_Ventilation_System_Manager;
    L_i : INT;
    L_Supply_Fans_Byte : ARRAY[1..GVL_CONSTANTS.C_MAX_SUPPLY_FANS] OF BYTE;
    L_Exhaust_Fans_Byte : ARRAY[1..GVL_CONSTANTS.C_MAX_EXHAUST_FANS] OF BYTE;
    L_Wet_Zone_Active : ARRAY[1..GVL_CONSTANTS.C_MAX_WET_ZONES] OF BOOL;
    L_Vent_PV3_Boost_Req : BOOL;
    L_Supply_100_Req : BOOL;
    L_Exhaust_100_Req : BOOL;
    L_Supply_80_Req : BOOL;
    L_Vent_Stop_Req : BOOL;
  END_VAR

            // Wet-zone adapter
FOR L_i := 1 TO GVL_CONSTANTS.C_MAX_WET_ZONES DO
    L_Wet_Zone_Active[L_i] := FALSE;
END_FOR;
IF GVL_STATUS.G_Wet_Zone_Light_Active THEN
    L_Wet_Zone_Active[1] := TRUE;
END_IF;

// === Ventilation Inputs (from arbitration only) ===
L_Vent_PV3_Boost_Req := GVL_COMMAND_SHADOW.G_Vent_PV3_Boost;
L_Supply_100_Req := GVL_COMMAND_SHADOW.G_Supply_100_Req;
L_Exhaust_100_Req := GVL_COMMAND_SHADOW.G_Exhaust_100_Req;
L_Supply_80_Req := GVL_COMMAND_SHADOW.G_Supply_80_Req;
L_Vent_Stop_Req := GVL_COMMAND_SHADOW.G_Vent_Stop;

// Coordinator constraint: block non-stop ventilation requests only.
// Safety-driven stop request must remain untouched.
IF GVL_SYSTEM_COORDINATION.G_Block_Ventilation THEN
    L_Vent_PV3_Boost_Req := FALSE;
    L_Supply_100_Req := FALSE;
    L_Exhaust_100_Req := FALSE;
    L_Supply_80_Req := FALSE;
END_IF;

// 11. Управление вентиляцией
fbVentilationManager(
    VI_System_Time_MS := GVL_STATUS.G_System_Time_MS,
    VI_IsActivePLC := GVL_STATUS.G_Is_Active_PLC,
    VI_Outdoor_Temp := GVL_STATE.G_Outdoor_Temp,
    VI_Supply_Temps := GVL_STATE.G_Supply_Temps,
    VI_Room_Temps := GVL_STATE.G_Room_Temps,
    VI_Room_Humidities := GVL_STATE.G_Room_Hum,
    VI_Room_CO2 := GVL_STATE.G_Room_CO2,
    VI_Current_Scenario := GVL_STATUS.G_Current_Scenario,
    VI_System_Mode := GVL_STATE.G_System_Mode,
    VI_Config := GVL_CONFIG.G_HMI_Vent_Global_Config,
    VI_Fire_Alarm := GVL_STATE.G_Safety_Smoke_Latched,
    VI_Gas_Alarm := GVL_STATE.G_Safety_Gas_Latched,
    VI_PV3_Boost_Req := L_Vent_PV3_Boost_Req,
    VI_Supply_100_Req := L_Supply_100_Req,
    VI_Exhaust_100_Req := L_Exhaust_100_Req,
    VI_Supply_80_Req := L_Supply_80_Req,
    VI_Vent_Stop := L_Vent_Stop_Req,
    VI_IO_Modules_Online := GVL_STATUS.G_IO_Modules_Online,
    VI_Wet_Zone_Active := L_Wet_Zone_Active,
    VI_Rule_Actions := GVL_STATE.G_Rule_Actions,
    VO_Supply_Fans => L_Supply_Fans_Byte,
    VO_Exhaust_Fans => L_Exhaust_Fans_Byte,
    VO_Heater_Power => GVL_STATE.G_Vent_Heater_Power,
    VO_Status_Msg => GVL_STATUS.G_Vent_Status_Msg,
    VO_Ventilation_IO_Fault => GVL_STATE.G_Ventilation_IO_Fault,
    VO_Ventilation_Subsystem_Degraded => GVL_STATE.G_Ventilation_Subsystem_Degraded
);
// >>> BULK_SYNC_ANCHOR: PRG_Ventilation <<<


// Ventilation copy-out adapters
FOR L_i := 1 TO GVL_CONSTANTS.C_MAX_SUPPLY_FANS DO
    GVL_STATE.G_Supply_Fans[L_i] := BYTE_TO_REAL(L_Supply_Fans_Byte[L_i]);
END_FOR;
FOR L_i := 1 TO GVL_CONSTANTS.C_MAX_EXHAUST_FANS DO
    GVL_STATE.G_Exhaust_Fans[L_i] := BYTE_TO_REAL(L_Exhaust_Fans_Byte[L_i]);
END_FOR;
          
END_PROGRAM

PROGRAM PRG_PLC_A

            // Вызов основной программы
PRG_System();
// >>> BULK_SYNC_ANCHOR: PRG_PLC_A <<<
          
END_PROGRAM

PROGRAM PRG_Command_Verifier
  VAR
    L_Mismatch_Count : INT := 0;
  END_VAR

            // Current-cycle mismatch count between legacy and shadow command layers
L_Mismatch_Count := 0;

IF GVL_COMMAND.G_Gas_Valve_Close <> GVL_COMMAND_SHADOW.G_Gas_Valve_Close THEN
    L_Mismatch_Count := L_Mismatch_Count + 1;
END_IF;

IF GVL_COMMAND.G_Boiler_Stop <> GVL_COMMAND_SHADOW.G_Boiler_Stop THEN
    L_Mismatch_Count := L_Mismatch_Count + 1;
END_IF;

IF GVL_COMMAND.G_Vent_Stop <> GVL_COMMAND_SHADOW.G_Vent_Stop THEN
    L_Mismatch_Count := L_Mismatch_Count + 1;
END_IF;

IF GVL_COMMAND.G_Supply_100_Req <> GVL_COMMAND_SHADOW.G_Supply_100_Req THEN
    L_Mismatch_Count := L_Mismatch_Count + 1;
END_IF;

IF GVL_COMMAND.G_Supply_80_Req <> GVL_COMMAND_SHADOW.G_Supply_80_Req THEN
    L_Mismatch_Count := L_Mismatch_Count + 1;
END_IF;

IF GVL_COMMAND.G_Vent_PV3_Boost <> GVL_COMMAND_SHADOW.G_Vent_PV3_Boost THEN
    L_Mismatch_Count := L_Mismatch_Count + 1;
END_IF;

IF GVL_COMMAND.G_Close_Valve_35 <> GVL_COMMAND_SHADOW.G_Close_Valve_35 THEN
    L_Mismatch_Count := L_Mismatch_Count + 1;
END_IF;

IF GVL_COMMAND.G_Close_Valve_36 <> GVL_COMMAND_SHADOW.G_Close_Valve_36 THEN
    L_Mismatch_Count := L_Mismatch_Count + 1;
END_IF;

IF GVL_COMMAND.G_Lock_1_Open <> GVL_COMMAND_SHADOW.G_Lock_1_Open THEN
    L_Mismatch_Count := L_Mismatch_Count + 1;
END_IF;

IF GVL_COMMAND.G_Lock_1_Close <> GVL_COMMAND_SHADOW.G_Lock_1_Close THEN
    L_Mismatch_Count := L_Mismatch_Count + 1;
END_IF;

IF GVL_COMMAND.G_Lock_2_Open <> GVL_COMMAND_SHADOW.G_Lock_2_Open THEN
    L_Mismatch_Count := L_Mismatch_Count + 1;
END_IF;

IF GVL_COMMAND.G_Lock_2_Close <> GVL_COMMAND_SHADOW.G_Lock_2_Close THEN
    L_Mismatch_Count := L_Mismatch_Count + 1;
END_IF;

// Gate and wicket comparison
IF GVL_COMMAND.G_Gate_Open <> GVL_COMMAND_SHADOW.G_Gate_Open THEN
    L_Mismatch_Count := L_Mismatch_Count + 1;
END_IF;

IF GVL_COMMAND.G_Wicket_Open <> GVL_COMMAND_SHADOW.G_Wicket_Open THEN
    L_Mismatch_Count := L_Mismatch_Count + 1;
END_IF;

GVL_COMMAND_VERIFY.Command_Mismatch_Count := L_Mismatch_Count;
GVL_COMMAND_VERIFY.Command_Match_OK := (L_Mismatch_Count = 0);
GVL_COMMAND_VERIFY.Command_Mismatch_Active := (L_Mismatch_Count > 0);
          
END_PROGRAM

PROGRAM PRG_Heating_Policy_Observer
  VAR
    fbPolicy : FB_Heating_Policy_Observer;
  END_VAR

            fbPolicy(
    VI_Zone_Occupied := GVL_PRESENCE.G_Zone_Occupied,
    VI_Zone_Last_Motion_TS := GVL_PRESENCE.G_Zone_Last_Motion_TS,
    VI_System_Time_MS := GVL_STATUS.G_System_Time_MS,
    VI_Zone_Permanent_Use := GVL_HEATING_POLICY.G_Zone_Permanent_Use,
    VI_Zone_Guest_Preheat := GVL_HEATING_POLICY.G_Zone_Guest_Preheat_Request,
    VI_Behavior_Mode := GVL_MODE.G_Current_Behavior_Mode
);

GVL_HEATING_POLICY.G_Zone_Empty_Duration_MS := fbPolicy.VO_Zone_Empty_Duration_MS;
GVL_HEATING_POLICY.G_Zone_Policy_Class := fbPolicy.VO_Zone_Policy_Class;
GVL_HEATING_POLICY.G_Zone_Target_Adjustment := fbPolicy.VO_Zone_Target_Adjustment;
GVL_HEATING_POLICY.G_Zone_Priority_Bias := fbPolicy.VO_Zone_Priority_Bias;
          
END_PROGRAM

PROGRAM PLC_PRG

            // Вызов основных программ
PRG_IO_Read();
PRG_Safety();
PRG_System();
PRG_Presence_Manager();
PRG_Heating_Policy_Observer();
PRG_Mode_Manager();
PRG_System_Coordinator();
PRG_Policy();
PRG_Command_Arbitration();
PRG_Command_Verifier();
PRG_Security();
PRG_Heating();
PRG_Ventilation();
PRG_Lighting();
PRG_IO_Write();

// PRG_Test(); // Раскомментировать для запуска модульных тестов
          
END_PROGRAM
